TYPE ST_SurrenderHands :
STRUCT
	//Player has a 15 and dealer is showing a 10
	//Player has a 16 and dealer is showing a 9, 10 or A
END_STRUCT
END_TYPE

(* stored: Version 1.1.0.1, ProductVersion 3.1.4024.10
   DUT ST_SurrenderHands: Id {79a0a2ab-dc75-47aa-9327-bd58006616e8} *)
